FUNCTION TFPackCodePresenteInZona_old : INT
VAR_INPUT
	//HandlingPackTable : POINTER TO TFHandlingPackTable;
	ArrayPacchi : POINTER TO DUT_ArrayPacchi;
	WorkAreaZone : POINTER TO TFMachinePalletizer_WorkAreaZone;
	WorkArea : INT;
END_VAR
VAR
	w : INT;
	n : INT;
	i : INT;
	a : INT;
END_VAR

TFPackCodePresenteInZona := 0; 

//FOR w:=1 TO MAXDIMARRAYPACCHI DO
	IF ArrayPacchi^.Pacco[1].PC > 0 THEN
		FOR n:=1 TO MAXZONE DO
			FOR a:=1 TO MAXAREA DO
				IF WorkAreaZone^.Zone[n].WorkArea[a] = WorkArea THEN
					FOR i:=1 TO MAXFORMINGCODE DO
						(* Verifico se il Pacco presente nel WPP è destinato ad una Zona *)
						IF WorkAreaZone^.Zone[n].Code[i] = ArrayPacchi^.Pacco[1].PC THEN
							TFPackCodePresenteInZona := ArrayPacchi^.Pacco[w].PC;
							RETURN;
						END_IF
					END_FOR
				END_IF
			END_FOR
		END_FOR
	END_IF
//END_FOR

END_FUNCTION

(* stored: Version 1.1.0.1, ProductVersion 3.1.4024.11
   POU TFPackCodePresenteInZona_old: Id {9f5d154a-dcfc-47e6-b928-f4c8d08eb469}, SpecialFunc None *)
